(* LS Electric XG5000 project: 241004_실습4_모터작동내부변수사용 *)
(* PLC LSPLC *)

PROGRAM NewProgram (* task: 스캔 프로그램 *)
VAR
    PB0 AT %IX0.0.0 : BOOL;
    PB1 AT %IX0.0.1 : BOOL;
    내부변수 AT %MX0 : BOOL;
    모터1 AT %QX0.1.0 : BOOL;
    모터2 AT %QX0.1.1 : BOOL;
    모터3 AT %QX0.1.2 : BOOL;
END_VAR
VAR
    _e1 : R_TRIG;
    _e2 : R_TRIG;
END_VAR

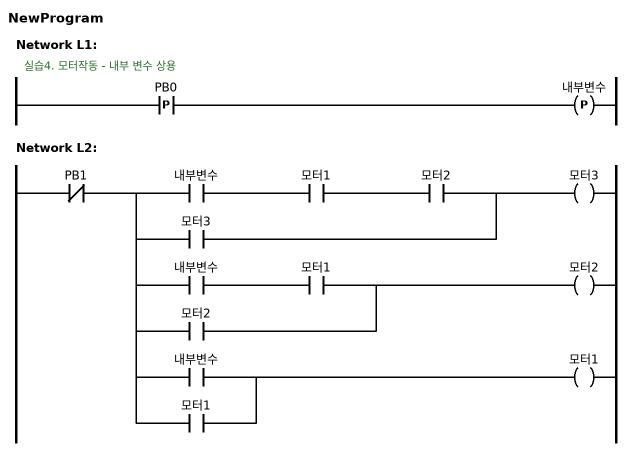
(* 실습4. 모터작동 - 내부 변수 상용 *)
(* Rung L1 *)
_e1(CLK := PB0);
_e2(CLK := _e1.Q);
내부변수 := _e2.Q;
(* Rung L2 *)
모터3 := NOT PB1 AND ((내부변수 AND 모터1 AND 모터2) OR 모터3);
모터2 := NOT PB1 AND ((내부변수 AND 모터1) OR 모터2);
모터1 := NOT PB1 AND (내부변수 OR 모터1);
END_PROGRAM